	IF
	// NX5001_2
		DiagsRetain.DG_NX5001_2_tGeneral_bActiveDiagnostics OR
		DiagsRetain.DG_NX5001_2_tGeneral_bBusCommunicationError OR
		DiagsRetain.DG_NX5001_2_tGeneral_bConfigMismatch OR
		DiagsRetain.DG_NX5001_2_tGeneral_bFatalError OR
		DiagsRetain.DG_NX5001_2_tGeneral_bNX5001NoCfg OR
		DiagsRetain.DG_NX5001_2_tGeneral_bOTDSwitchError OR
		DiagsRetain.DG_NX5001_2_tGeneral_bPbusCommFail OR
		DiagsRetain.DG_NX5001_2_tGeneral_bSlaveNotConfigured OR
		DiagsRetain.DG_NX5001_2_tGeneral_bSlaveNotPresent OR
		DiagsRetain.DG_NX5001_2_tGeneral_bSlaveWithDiagnostic OR
		DiagsRetain.DG_NX5001_2_tGeneral_bStsEnableInterface OR
	//	DiagsRetain.DG_NX5001_2_tGeneral_bStsMstRedundEnable OR   Demanda 17571
		DiagsRetain.DG_NX5001_2_tGeneral_bWatchdogError THEN
   	 	bDiag_Error_NX5001_2:= TRUE;
	ELSE
		bDiag_Error_NX5001_2:= FALSE;	
	END_IF
	
	IF
	// NX5001_3
		DiagsRetain.DG_NX5001_3_tGeneral_bActiveDiagnostics OR
		DiagsRetain.DG_NX5001_3_tGeneral_bBusCommunicationError OR
		DiagsRetain.DG_NX5001_3_tGeneral_bConfigMismatch OR
		DiagsRetain.DG_NX5001_3_tGeneral_bFatalError OR
		DiagsRetain.DG_NX5001_3_tGeneral_bNX5001NoCfg OR
		DiagsRetain.DG_NX5001_3_tGeneral_bOTDSwitchError OR
		DiagsRetain.DG_NX5001_3_tGeneral_bPbusCommFail OR
		DiagsRetain.DG_NX5001_3_tGeneral_bSlaveNotConfigured OR
		DiagsRetain.DG_NX5001_3_tGeneral_bSlaveNotPresent OR
		DiagsRetain.DG_NX5001_3_tGeneral_bSlaveWithDiagnostic OR
		DiagsRetain.DG_NX5001_3_tGeneral_bStsEnableInterface OR
	//	DiagsRetain.DG_NX5001_3_tGeneral_bStsMstRedundEnable OR   Demanda 17571
		DiagsRetain.DG_NX5001_3_tGeneral_bWatchdogError THEN
  	 	bDiag_Error_NX5001_3:= TRUE;
	ELSE
		bDiag_Error_NX5001_3:= FALSE;	
	END_IF
	
	IF
	// NX5000_1	
		DiagsRetain.DG_NX5000_1_tGeneral_bActiveDiagnostics OR
		DiagsRetain.DG_NX5000_1_tGeneral_bBusCommunicationError OR
		DiagsRetain.DG_NX5000_1_tGeneral_bConfigMismatch OR
		DiagsRetain.DG_NX5000_1_tGeneral_bFatalError OR
		DiagsRetain.DG_NX5000_1_tGeneral_bOTDSwitchError OR
		DiagsRetain.DG_NX5000_1_tGeneral_bWatchdogError OR
		DiagsRetain.DG_NX5000_1_tNX5000_bNX5000NoCfg OR
		DiagsRetain.DG_NX5000_1_tNX5000_bStsEthLink THEN
    	bDiag_Error_NX5000_1:= TRUE;
	ELSE
		bDiag_Error_NX5000_1:= FALSE;	
	END_IF
	
	IF
	// NX5000_2	
		DiagsRetain.DG_NX5000_2_tGeneral_bActiveDiagnostics OR
		DiagsRetain.DG_NX5000_2_tGeneral_bBusCommunicationError OR
		DiagsRetain.DG_NX5000_2_tGeneral_bConfigMismatch OR
		DiagsRetain.DG_NX5000_2_tGeneral_bFatalError OR
		DiagsRetain.DG_NX5000_2_tGeneral_bOTDSwitchError OR
		DiagsRetain.DG_NX5000_2_tGeneral_bWatchdogError OR
		DiagsRetain.DG_NX5000_2_tNX5000_bNX5000NoCfg OR
		DiagsRetain.DG_NX5000_2_tNX5000_bStsEthLink THEN
    	bDiag_Error_NX5000_2:= TRUE;
	ELSE
		bDiag_Error_NX5000_2:= FALSE;	
	END_IF
	
	IF
	// NX5000_3	
		DiagsRetain.DG_NX5000_3_tGeneral_bActiveDiagnostics OR
		DiagsRetain.DG_NX5000_3_tGeneral_bBusCommunicationError OR
		DiagsRetain.DG_NX5000_3_tGeneral_bConfigMismatch OR
		DiagsRetain.DG_NX5000_3_tGeneral_bFatalError OR
		DiagsRetain.DG_NX5000_3_tGeneral_bOTDSwitchError OR
		DiagsRetain.DG_NX5000_3_tGeneral_bWatchdogError OR
		DiagsRetain.DG_NX5000_3_tNX5000_bNX5000NoCfg OR
		DiagsRetain.DG_NX5000_3_tNX5000_bStsEthLink THEN
    	bDiag_Error_NX5000_3:= TRUE;
	ELSE
		bDiag_Error_NX5000_3:= FALSE;	
	END_IF
	
	IF
	// DiagsRetain.DG_MODBUS_Master_1
		DiagsRetain.DG_MODBUS_Master_1_tDiag_bConfigFailure OR
		DiagsRetain.DG_MODBUS_Master_1_tDiag_bModuleFailure OR
		DiagsRetain.DG_MODBUS_Master_1_tDiag_bRXFailure OR
		DiagsRetain.DG_MODBUS_Master_1_tDiag_bTXFailure THEN
   	 	bDiag_Error_MODBUS_Master_1:= TRUE;
	ELSE
		bDiag_Error_MODBUS_Master_1:= FALSE;	
	END_IF
	
	IF
	// MODBUS_Slave_1	
		DiagsRetain.DG_MODBUS_Slave_1_tDiag_bConfigFailure OR
		DiagsRetain.DG_MODBUS_Slave_1_tDiag_bModuleFailure OR
		DiagsRetain.DG_MODBUS_Slave_1_tDiag_bRXFailure OR
		DiagsRetain.DG_MODBUS_Slave_1_tDiag_bTXFailure THEN
   		bDiag_Error_MODBUS_Slave_1:= TRUE;
	ELSE
		bDiag_Error_MODBUS_Slave_1:= FALSE;	
	END_IF
	
	IF
	// MODBUS_Client_2
		DiagsRetain.DG_MODBUS_Client_2_tDiag_bConfigFailure OR
//		DiagsRetain.DG_MODBUS_Client_2_tDiag_bModuleFailure OR 	// Demanda 13816
		DiagsRetain.DG_MODBUS_Client_2_tDiag_bRXFailure OR
		DiagsRetain.DG_MODBUS_Client_2_tDiag_bTXFailure THEN
    	bDiag_Error_MODBUS_Client_2:= TRUE;
	ELSE
		bDiag_Error_MODBUS_Client_2:= FALSE;	
	END_IF
	
	IF
	// MODBUS_Server_2
		DiagsRetain.DG_MODBUS_Server_2_tDiag_bConfigFailure OR
		DiagsRetain.DG_MODBUS_Server_2_tDiag_bModuleFailure OR
		DiagsRetain.DG_MODBUS_Server_2_tDiag_bRXFailure OR
		DiagsRetain.DG_MODBUS_Server_2_tDiag_bTXFailure THEN
    	bDiag_Error_MODBUS_Server_2:= TRUE;
	ELSE
		bDiag_Error_MODBUS_Server_2:= FALSE;	
	END_IF
	
	IF
	// MODBUS_Client_3
		DiagsRetain.DG_MODBUS_Client_3_tDiag_bConfigFailure OR
		DiagsRetain.DG_MODBUS_Client_3_tDiag_bModuleFailure OR
		DiagsRetain.DG_MODBUS_Client_3_tDiag_bRXFailure OR
		DiagsRetain.DG_MODBUS_Client_3_tDiag_bTXFailure THEN
    	bDiag_Error_MODBUS_Client_3:= TRUE;
	ELSE
		bDiag_Error_MODBUS_Client_3:= FALSE;	
	END_IF
	
	IF
	// MODBUS_Server_3
		DiagsRetain.DG_MODBUS_Server_3_tDiag_bConfigFailure OR
//		DiagsRetain.DG_MODBUS_Server_3_tDiag_bModuleFailure OR  	// Demanda 13816
		DiagsRetain.DG_MODBUS_Server_3_tDiag_bRXFailure OR
		DiagsRetain.DG_MODBUS_Server_3_tDiag_bTXFailure THEN
    	bDiag_Error_MODBUS_Server_3:= TRUE;
	ELSE
		bDiag_Error_MODBUS_Server_3:= FALSE;	
	END_IF
	
	IF
	// MODBUS_Client_4
		DiagsRetain.DG_MODBUS_Client_4_tDiag_bConfigFailure OR
		DiagsRetain.DG_MODBUS_Client_4_tDiag_bModuleFailure OR
		DiagsRetain.DG_MODBUS_Client_4_tDiag_bRXFailure OR
		DiagsRetain.DG_MODBUS_Client_4_tDiag_bTXFailure THEN
    	bDiag_Error_MODBUS_Client_4:= TRUE;
	ELSE
		bDiag_Error_MODBUS_Client_4:= FALSE;	
	END_IF
	
	IF
	// MODBUS_Server_4	
		DiagsRetain.DG_MODBUS_Server_4_tDiag_bConfigFailure OR
//		DiagsRetain.DG_MODBUS_Server_4_tDiag_bModuleFailure OR  	// Demanda 13816
		DiagsRetain.DG_MODBUS_Server_4_tDiag_bRXFailure OR
		DiagsRetain.DG_MODBUS_Server_4_tDiag_bTXFailure THEN
    	bDiag_Error_MODBUS_Server_4:= TRUE;
	ELSE
		bDiag_Error_MODBUS_Server_4:= FALSE;	
	END_IF
	

	IF		
		//PO1000
		DiagsRetain.DG_REM05_PO1000_bHardwareFailure OR
		DiagsRetain.DG_REM05_PO1000_bPowerSupplyFail THEN
	   	bDiag_Error_PO1000_REM05:= TRUE;
	ELSE
		bDiag_Error_PO1000_REM05:= FALSE;	
	END_IF
	
	IF		
		//PO2020
		DiagsRetain.DG_REM05_PO2020_bHardwareFailure OR
		DiagsRetain.DG_REM05_PO2020_bPowerSupplyFail THEN
		bDiag_Error_PO2020_REM05:= TRUE;
	ELSE
		bDiag_Error_PO2020_REM05:= FALSE;	
	END_IF

	IF		
		//PO9100	
		DiagsRetain.DG_REM05_PO9100_bReserved00 THEN
		bDiag_Error_PO9100_REM05:= TRUE;
	ELSE
		bDiag_Error_PO9100_REM05:= FALSE;	
	END_IF	
	
	IF		
	//PO1212
	DiagsRetain.DG_REM10_PO1212_bFuseOpen OR
	DiagsRetain.DG_REM10_PO1212_bHardwareFailure OR
	DiagsRetain.DG_REM10_PO1212_bNoParametrizedModule OR
	DiagsRetain.DG_REM10_PO1212_bOverTemp OR
	DiagsRetain.DG_REM10_PO1212_aCh0_bOpenSensor OR
	DiagsRetain.DG_REM10_PO1212_aCh0_bOverRange OR
	DiagsRetain.DG_REM10_PO1212_aCh0_bSensorShortCircuit OR
	DiagsRetain.DG_REM10_PO1212_aCh0_bWrongParameters OR
	DiagsRetain.DG_REM10_PO1212_aCh1_bOpenSensor OR
	DiagsRetain.DG_REM10_PO1212_aCh1_bOverRange OR
	DiagsRetain.DG_REM10_PO1212_aCh1_bSensorShortCircuit OR
	DiagsRetain.DG_REM10_PO1212_aCh1_bWrongParameters OR
	DiagsRetain.DG_REM10_PO1212_aCh2_bOpenSensor OR
	DiagsRetain.DG_REM10_PO1212_aCh2_bOverRange OR
	DiagsRetain.DG_REM10_PO1212_aCh2_bSensorShortCircuit OR
	DiagsRetain.DG_REM10_PO1212_aCh2_bWrongParameters OR
	DiagsRetain.DG_REM10_PO1212_aCh3_bOpenSensor OR
	DiagsRetain.DG_REM10_PO1212_aCh3_bOverRange OR
	DiagsRetain.DG_REM10_PO1212_aCh3_bSensorShortCircuit OR
	DiagsRetain.DG_REM10_PO1212_aCh3_bWrongParameters OR
	DiagsRetain.DG_REM10_PO1212_aCh4_bOpenSensor OR
	DiagsRetain.DG_REM10_PO1212_aCh4_bOverRange OR
	DiagsRetain.DG_REM10_PO1212_aCh4_bSensorShortCircuit OR
	DiagsRetain.DG_REM10_PO1212_aCh4_bWrongParameters OR
	DiagsRetain.DG_REM10_PO1212_aCh5_bOpenSensor OR
	DiagsRetain.DG_REM10_PO1212_aCh5_bOverRange OR
	DiagsRetain.DG_REM10_PO1212_aCh5_bSensorShortCircuit OR
	DiagsRetain.DG_REM10_PO1212_aCh5_bWrongParameters OR
	DiagsRetain.DG_REM10_PO1212_aCh6_bOpenSensor OR
	DiagsRetain.DG_REM10_PO1212_aCh6_bOverRange OR
	DiagsRetain.DG_REM10_PO1212_aCh6_bSensorShortCircuit OR
	DiagsRetain.DG_REM10_PO1212_aCh6_bWrongParameters OR
	DiagsRetain.DG_REM10_PO1212_aCh7_bOpenSensor OR
	DiagsRetain.DG_REM10_PO1212_aCh7_bOverRange OR
	DiagsRetain.DG_REM10_PO1212_aCh7_bSensorShortCircuit OR
	DiagsRetain.DG_REM10_PO1212_aCh7_bWrongParameters THEN
		bDiag_Error_PO1212_REM10:= TRUE;
	ELSE
		bDiag_Error_PO1212_REM10:= FALSE;	
	END_IF		
	
	IF		
	//PO2132
	DiagsRetain.DG_REM10_PO2132_bNoParametrizedModule OR
	DiagsRetain.DG_REM10_PO2132_bPowerSupplyFail OR
	DiagsRetain.DG_REM10_PO2132_aCh0_bOpenSensor OR
	DiagsRetain.DG_REM10_PO2132_aCh0_bWrongParameters OR
	DiagsRetain.DG_REM10_PO2132_aCh1_bOpenSensor OR
	DiagsRetain.DG_REM10_PO2132_aCh1_bWrongParameters OR
	DiagsRetain.DG_REM10_PO2132_aCh2_bOpenSensor OR
	DiagsRetain.DG_REM10_PO2132_aCh2_bWrongParameters OR
	DiagsRetain.DG_REM10_PO2132_aCh3_bOpenSensor OR
	DiagsRetain.DG_REM10_PO2132_aCh3_bWrongParameters THEN
		bDiag_Error_PO2132_REM10:= TRUE;
	ELSE
		bDiag_Error_PO2132_REM10:= FALSE;	
	END_IF		
	
	IF		
	//PO9100
	DiagsRetain.DG_REM10_PO9100_bReserved00 THEN
			bDiag_Error_PO9100_REM10:= TRUE;
	ELSE
		bDiag_Error_PO9100_REM10:= FALSE;	
	END_IF	
	
	IF		
	//PO1000
	DiagsRetain.DG_REM04_PO1000_bHardwareFailure OR
	DiagsRetain.DG_REM04_PO1000_bPowerSupplyFail THEN
		bDiag_Error_PO1000_REM04:= TRUE;
	ELSE
		bDiag_Error_PO1000_REM04:= FALSE;	
	END_IF	

	
	IF 
		bDiag_Error_NX3030 OR
		bDiag_Error_NX4010 OR
		bDiag_Error_NX5001_1 OR
		bDiag_Error_NX5001_2 OR
		bDiag_Error_NX5001_3 OR
		bDiag_Error_NX5000_1 OR
		bDiag_Error_NX5000_2 OR
		bDiag_Error_NX5000_3 OR
		bDiag_Error_MODBUS_Master_1 OR
		bDiag_Error_MODBUS_Slave_1 OR
		bDiag_Error_MODBUS_Client_2 OR
		bDiag_Error_MODBUS_Server_2 OR
		bDiag_Error_MODBUS_Client_3 OR
		bDiag_Error_MODBUS_Server_3 OR
		bDiag_Error_MODBUS_Client_4 OR
		bDiag_Error_MODBUS_Server_4 OR	
		bDiag_Error_PO1000_REM05 OR
		bDiag_Error_PO2020_REM05 OR
		bDiag_Error_PO9100_REM05 OR
		bDiag_Error_PO1212_REM10 OR
		bDiag_Error_PO2132_REM10 OR
		bDiag_Error_PO9100_REM10 OR
		bDiag_Error_PO1000_REM04 THEN
		PersistentVars.bActiveDiagPlcB:= TRUE;
	ELSE
		PersistentVars.bActiveDiagPlcB:= FALSE;
	END_IF
END_IF	

// Limpa diagnóstico com um comando de CleanTest
IF SymbolicsNonRedundant.bEnableCleanStats_CheckDiagsRetain THEN
	SymbolicsNonRedundant.bEnableCleanStats_CheckDiagsRetain:= FALSE;
	PersistentVars.bActiveDiagPlcB:= FALSE;
	PersistentVars.bActiveDiagPlcA:= FALSE;
	/// Depuração 1
	auiDebugRedDataSync[0]:= auiDebugRedForceSync[0]:= 0;
	auiDebugRedDataSync[1]:= auiDebugRedForceSync[1]:= 0;
	auiDebugRedDataSync[2]:= auiDebugRedForceSync[2]:= 0;
	auiDebugRedDataSync[3]:= auiDebugRedForceSync[3]:= 0;
	auiDebugRedDataSync[4]:= auiDebugRedForceSync[4]:= 0;
	auiDebugRedDataSync[5]:= auiDebugRedForceSync[5]:= 0;
	auiDebugRedDataSync[6]:= auiDebugRedForceSync[6]:= 0;
END_IF

/// Depuração 2
IF NOT DG_NX4010.tRedundancy.RedDgnLoc.sGeneral_Diag.bRedDataSync THEN
	CASE fbRedundancyManagement.m_fbDiagnosticsLocal.eRedState OF
		REDUNDANCY_STATE.NOT_CONFIGURED:	auiDebugRedDataSync[0]:= MIN(auiDebugRedDataSync[0] + 1, 65000);
		REDUNDANCY_STATE.INIT:				auiDebugRedDataSync[1]:= MIN(auiDebugRedDataSync[1] + 1, 65000);
		REDUNDANCY_STATE.STARTING:			auiDebugRedDataSync[2]:= MIN(auiDebugRedDataSync[2] + 1, 65000);
		REDUNDANCY_STATE.STANDBY:			auiDebugRedDataSync[3]:= MIN(auiDebugRedDataSync[3] + 1, 65000);
		REDUNDANCY_STATE.ACTIVE:			auiDebugRedDataSync[4]:= MIN(auiDebugRedDataSync[4] + 1, 65000);
		REDUNDANCY_STATE.INACTIVE:			auiDebugRedDataSync[5]:= MIN(auiDebugRedDataSync[5] + 1, 65000);
	ELSE
		auiDebugRedDataSync[6]:= MIN(auiDebugRedDataSync[6] + 1, 65000);
	END_CASE
END_IF

/// Depuração 3
IF NOT DG_NX4010.tRedundancy.RedDgnLoc.sGeneral_Diag.bRedForceSync THEN
	CASE fbRedundancyManagement.m_fbDiagnosticsLocal.eRedState OF
		REDUNDANCY_STATE.NOT_CONFIGURED:	auiDebugRedForceSync[0]:= MIN(auiDebugRedForceSync[0] + 1, 65000);
		REDUNDANCY_STATE.INIT:				auiDebugRedForceSync[1]:= MIN(auiDebugRedForceSync[1] + 1, 65000);
		REDUNDANCY_STATE.STARTING:			auiDebugRedForceSync[2]:= MIN(auiDebugRedForceSync[2] + 1, 65000);
		REDUNDANCY_STATE.STANDBY:			auiDebugRedForceSync[3]:= MIN(auiDebugRedForceSync[3] + 1, 65000);
		REDUNDANCY_STATE.ACTIVE:			auiDebugRedForceSync[4]:= MIN(auiDebugRedForceSync[4] + 1, 65000);
		REDUNDANCY_STATE.INACTIVE:			auiDebugRedForceSync[5]:= MIN(auiDebugRedForceSync[5] + 1, 65000);
	ELSE
		auiDebugRedForceSync[6]:= MIN(auiDebugRedForceSync[6] + 1, 65000);
	END_CASE
END_IF

// Registra o tempo do sistema
SysTimeGetUs(uliPouEndTime);
// Calcula duração mínima/máxima desta POU
MinMaxTimes.uliPouMinTime_CheckDiags:= MIN(MinMaxTimes.uliPouMinTime_CheckDiags, uliPouEndTime - uliPouIniTime);
MinMaxTimes.uliPouMaxTime_CheckDiags:= MAX(MinMaxTimes.uliPouMaxTime_CheckDiags, uliPouEndTime - uliPouIniTime);

END_PROGRAM

// Device/Application/UserPOUs/Non-Redundant/DaylightSavingTime
PROGRAM DaylightSavingTime
VAR
	xDateAndTime:	EXTENDED_DATE_AND_TIME;
	byDayOfWeek:	BYTE;
	xTimeZoneRd:	TIMEZONESETTINGS;
	xTimeZoneWr:	TIMEZONESETTINGS;
	// Array de referência para cada ano:
	// 14 indica que o terceiro domingo do mês de fevereiro NÃO coincide com o carnaval
	// 21 indica que o terceiro domingo do mês de fevereiro coincide com o carnaval
	aby3rd4thDay:	ARRAY[2017..2027] OF BYTE:= [14,14,14,14,14,14,21,14,14,21,14];
	// Contador de escritas do timezone em função do início/fim do horário de verão
	// (configurar o parâmetro "HX3040 > Synchronism > Time Zone" para o valor -3:00) 
	// (se iniciar a aplicação no horário de verão, o contador vai para 1 na partida) 
	udiTZWriteCnt:	UDINT;
	uliPouIniTime:	ULINT;
	uliPouEndTime:	ULINT;
END_VAR

// Rotina que detecta se é horário de verão, ajustando o timezone da UCP se necessário.

// Registra o tempo do sistema
SysTimeGetUs(uliPouIniTime);

// Leitura da data e hora atual, com sucesso...
IF NextoStandard.GetDateAndTime(xDateAndTime) = 0 THEN
	
	// Leitura do dia da semana
	byDayOfWeek:= NextoStandard.GetDayOfWeek();
	
	// Segundo o decreto presidencial 6.558 de 08/09/2008, o horário de verão inicia
	// no terceiro domingo do mês de outubro e termina no terceiro domingo do mês de
	// fevereiro (ou quarto, se o terceiro coincidir com a semana do carnaval)
	IF 	(xDateAndTime.byMonth = 10 AND (xDateAndTime.byDayOfMonth >= 14 + byDayOfWeek)) OR
		(xDateAndTime.byMonth = 11) OR
		(xDateAndTime.byMonth = 12) OR
		(xDateAndTime.byMonth = 1) OR
		(xDateAndTime.byMonth = 2 AND (xDateAndTime.byDayOfMonth < aby3rd4thDay[xDateAndTime.wYear] + byDayOfWeek)) THEN
			// Indica que é horário de verão
			NonRedData.bDaylightSavingTime:= TRUE;
	ELSE
			// Indica que NÃO é horário de verão
			NonRedData.bDaylightSavingTime:= FALSE;
	END_IF
	
	// Leitura do timezone, com sucesso...
	IF NextoStandard.GetTimeZone(xTimeZoneRd) = 0 THEN
		// Se horário de verão, timezone deve ser -2:00, caso contrário deve ser -3:00
		// Dispara um comando de escrita do timezone se encontrar alguma divergência
		IF 	(NonRedData.bDaylightSavingTime = TRUE AND (xTimeZoneRd.iHour <> -2 OR xTimeZoneRd.iMinutes <> 0)) OR
			(NonRedData.bDaylightSavingTime = FALSE AND (xTimeZoneRd.iHour <> -3 OR xTimeZoneRd.iMinutes <> 0)) THEN
				// Ajusta timezone para horário de verão ou horário normal
				IF NonRedData.bDaylightSavingTime = TRUE THEN
					xTimeZoneWr.iHour:= -2;
					xTimeZoneWr.iMinutes:= 0;
				ELSE
					xTimeZoneWr.iHour:= -3;
					xTimeZoneWr.iMinutes:= 0;
				END_IF
				// Chama função de escrita do timezone
				NextoStandard.SetTimeZone(xTimeZoneWr);
				// Incrementa o contador de escritas do timezone
				udiTZWriteCnt:= udiTZWriteCnt + 1;
		END_IF
	END_IF

END_IF

// Registra o tempo do sistema
SysTimeGetUs(uliPouEndTime);
// Calcula duração mínima/máxima desta POU
MinMaxTimes.uliPouMinTime_DaylightSavingTime:= MIN(MinMaxTimes.uliPouMinTime_DaylightSavingTime, uliPouEndTime - uliPouIniTime);
MinMaxTimes.uliPouMaxTime_DaylightSavingTime:= MAX(MinMaxTimes.uliPouMaxTime_DaylightSavingTime, uliPouEndTime - uliPouIniTime);

END_PROGRAM

// Device/Application/UserPOUs/Non-Redundant/CheckSpecialVarsRed
PROGRAM CheckSpecialVarsRed
VAR
	bPulse_100ms:		BOOL;
	bPulse_500ms:		BOOL;
	bPulse_1s:			BOOL;
	bPulse_2s:			BOOL;
	bPulse_5s:			BOOL;
	bPulse_10s:			BOOL;
	bPulse_30s:			BOOL;
	bPulse_60s:			BOOL;
	bPulse_Scan:		BOOL;
	
	di100msTimer:		DINT;
	di500msTimer:		DINT;
	di1sTimer:			DINT;
	di2sTimer:			DINT;
	di5sTimer:			DINT;
	di10sTimer:			DINT;
	di30sTimer:			DINT;
	di60sTimer:			DINT;
	
	bPulse100msFail:	BOOL;
	bPulse500msFail:	BOOL;
	bPulse1sFail:		BOOL;
	bPulse2sFail:		BOOL;
	bPulse5sFail:		BOOL;
	bPulse10sFail:		BOOL;
	bPulse30sFail:		BOOL;
	bPulse60sFail:		BOOL;
	bPulseScanFail:		BOOL;
	
	diMainTaskIntervalGapMs:	DINT:= ProjectConstants.iMainTaskInterval * 3 / 2;
	
	uliPouMemTime: 				ULINT;
	
END_VAR

// 
// POU para consistência das variáveis especiais redundantes.
// Esta POU deve ser chamada pela POU CheckSpecialVariables.
// 

// Detecta quando a tarefa cíclica deixou de ser chamada por um ciclo
// (com 10% de folga devido ao jitter negativo da tarefa)
// (também converte de milisegundos para microsegundos)
IF CheckSpecialVariables.uliPouIniTime > uliPouMemTime + DINT_TO_ULINT(ProjectConstants.iMainTaskInterval * 1900) THEN
	// Quando isso acontece, algumas variáveis de temporização e controle precisam ser ajustadas
	di100msTimer:= UDINT_TO_DINT(SpecialVariablesRedundantPrg.udiMicroAcc MOD 50000) / 1000;
	di500msTimer:= UDINT_TO_DINT(SpecialVariablesRedundantPrg.udiMicroAcc MOD 250000) / 1000;
	di1sTimer:= UDINT_TO_DINT(SpecialVariablesRedundantPrg.udiMicroAcc MOD 500000) / 1000;
	di2sTimer:= UDINT_TO_DINT(SpecialVariablesRedundantPrg.udiMicroAcc MOD 1000000) / 1000;
	di5sTimer:= UDINT_TO_DINT(SpecialVariablesRedundantPrg.udiMicroAcc MOD 2500000) / 1000;
	di10sTimer:= UDINT_TO_DINT(SpecialVariablesRedundantPrg.udiMicroAcc MOD 5000000) / 1000;
	di30sTimer:= UDINT_TO_DINT(SpecialVariablesRedundantPrg.udiMicroAcc MOD 15000000) / 1000;
	di60sTimer:= UDINT_TO_DINT(SpecialVariablesRedundantPrg.udiMicroAcc MOD 30000000) / 1000;
	bPulse_100ms:= Special_Variables_Redundant.Pulse_100ms_Redundant;
	bPulse_500ms:= Special_Variables_Redundant.Pulse_500ms_Redundant;
	bPulse_1s:= Special_Variables_Redundant.Pulse_1s_Redundant;
	bPulse_2s:= Special_Variables_Redundant.Pulse_2s_Redundant;
	bPulse_5s:= Special_Variables_Redundant.Pulse_5s_Redundant;
	bPulse_10s:= Special_Variables_Redundant.Pulse_10s_Redundant;
	bPulse_30s:= Special_Variables_Redundant.Pulse_30s_Redundant;
	bPulse_60s:= Special_Variables_Redundant.Pulse_60s_Redundant;
	bPulse_Scan:= NOT Special_Variables_Redundant.Pulse_Scan_Redundant;
END_IF
// Memoriza o tempo de ciclo atual
uliPouMemTime:= CheckSpecialVariables.uliPouIniTime;

// Executa parte do mesmo código que a SpecialVariablesRedundantPrg(), porém com variáveis locais:

	// Update scan pulse
	bPulse_Scan:= NOT bPulse_Scan;
	
// Mede e consiste a duração dos pulsos: frequência e duty-cycle (50%)

// Consiste o pulso de 100ms se o intervalo da tarefa não exceder os 33%
IF 100 > 3 * ProjectConstants.iMainTaskInterval THEN
	// Se o sinal não mudou de estado...
	IF bPulse_100ms = Special_Variables_Redundant.Pulse_100ms_Redundant THEN
		// Atualiza temporizador do sinal
		di100msTimer:= di100msTimer + ProjectConstants.iMainTaskInterval;
		// Indica erro caso o sinal não tenha mudado de estado no dobro do tempo esperado
		IF di100msTimer > 100 THEN bPulse100msFail:= TRUE; END_IF
	// Se o sinal mudou de estado...
	ELSE
		// Indica erro caso o sinal tenha mudado de estado antes ou depois do tempo esperado
		IF	di100msTimer < (100 / 2 - diMainTaskIntervalGapMs) OR
			di100msTimer > (100 / 2 + diMainTaskIntervalGapMs) THEN
				bPulse100msFail:= TRUE;
		END_IF
		// Inicializa o temporizador do sinal
		di100msTimer:= ProjectConstants.iMainTaskInterval;
		// Memoriza o estado atual do sinal
		bPulse_100ms:= Special_Variables_Redundant.Pulse_100ms_Redundant;
	END_IF
END_IF

// Consiste o pulso de 500ms se o intervalo da tarefa não exceder os 33%
IF 500 > 3 * ProjectConstants.iMainTaskInterval THEN
	// Se o sinal não mudou de estado...
	IF bPulse_500ms = Special_Variables_Redundant.Pulse_500ms_Redundant THEN
		// Atualiza temporizador do sinal
		di500msTimer:= di500msTimer + ProjectConstants.iMainTaskInterval;
		// Indica erro caso o sinal não tenha mudado de estado no dobro do tempo esperado
		IF di500msTimer > 500 THEN bPulse500msFail:= TRUE; END_IF
	// Se o sinal mudou de estado...
	ELSE
		// Indica erro caso o sinal tenha mudado de estado antes ou depois do tempo esperado
		IF	di500msTimer < (500 / 2 - diMainTaskIntervalGapMs) OR
			di500msTimer > (500 / 2 + diMainTaskIntervalGapMs) THEN
				bPulse500msFail:= TRUE;
		END_IF
		// Inicializa o temporizador do sinal
		di500msTimer:= ProjectConstants.iMainTaskInterval;
		// Memoriza o estado atual do sinal
		bPulse_500ms:= Special_Variables_Redundant.Pulse_500ms_Redundant;
	END_IF
END_IF

// Se o sinal não mudou de estado...
IF bPulse_1s = Special_Variables_Redundant.Pulse_1s_Redundant THEN
	// Atualiza temporizador do sinal
	di1sTimer:= di1sTimer + ProjectConstants.iMainTaskInterval;
	// Indica erro caso o sinal não tenha mudado de estado no dobro do tempo esperado
	IF di1sTimer > 1000 THEN bPulse1sFail:= TRUE; END_IF
// Se o sinal mudou de estado...
ELSE
	// Indica erro caso o sinal tenha mudado de estado antes ou depois do tempo esperado
	IF	di1sTimer < (1000 / 2 - diMainTaskIntervalGapMs) OR
		di1sTimer > (1000 / 2 + diMainTaskIntervalGapMs) THEN
			bPulse1sFail:= TRUE;
	END_IF
	// Inicializa o temporizador do sinal
	di1sTimer:= ProjectConstants.iMainTaskInterval;
	// Memoriza o estado atual do sinal
	bPulse_1s:= Special_Variables_Redundant.Pulse_1s_Redundant;
END_IF

// Se o sinal não mudou de estado...
IF bPulse_2s = Special_Variables_Redundant.Pulse_2s_Redundant THEN
	// Atualiza temporizador do sinal
	di2sTimer:= di2sTimer + ProjectConstants.iMainTaskInterval;
	// Indica erro caso o sinal não tenha mudado de estado no dobro do tempo esperado
	IF di2sTimer > 2000 THEN bPulse2sFail:= TRUE; END_IF
// Se o sinal mudou de estado...
ELSE
	// Indica erro caso o sinal tenha mudado de estado antes ou depois do tempo esperado
	IF	di2sTimer < (2000 / 2 - diMainTaskIntervalGapMs) OR
		di2sTimer > (2000 / 2 + diMainTaskIntervalGapMs) THEN
			bPulse2sFail:= TRUE;
	END_IF
	// Inicializa o temporizador do sinal
	di2sTimer:= ProjectConstants.iMainTaskInterval;
	// Memoriza o estado atual do sinal
	bPulse_2s:= Special_Variables_Redundant.Pulse_2s_Redundant;
END_IF

// Se o sinal não mudou de estado...
IF bPulse_5s = Special_Variables_Redundant.Pulse_5s_Redundant THEN
	// Atualiza temporizador do sinal
	di5sTimer:= di5sTimer + ProjectConstants.iMainTaskInterval;
	// Indica erro caso o sinal não tenha mudado de estado no dobro do tempo esperado
	IF di5sTimer > 5000 THEN bPulse5sFail:= TRUE; END_IF
// Se o sinal mudou de estado...
ELSE
	// Indica erro caso o sinal tenha mudado de estado antes ou depois do tempo esperado
	IF	di5sTimer < (5000 / 2 - diMainTaskIntervalGapMs) OR
		di5sTimer > (5000 / 2 + diMainTaskIntervalGapMs) THEN
			bPulse5sFail:= TRUE;
	END_IF
	// Inicializa o temporizador do sinal
	di5sTimer:= ProjectConstants.iMainTaskInterval;
	// Memoriza o estado atual do sinal
	bPulse_5s:= Special_Variables_Redundant.Pulse_5s_Redundant;
END_IF

// Se o sinal não mudou de estado...
IF bPulse_10s = Special_Variables_Redundant.Pulse_10s_Redundant THEN
	// Atualiza temporizador do sinal
	di10sTimer:= di10sTimer + ProjectConstants.iMainTaskInterval;
	// Indica erro caso o sinal não tenha mudado de estado no dobro do tempo esperado
	IF di10sTimer > 10000 THEN bPulse10sFail:= TRUE; END_IF
// Se o sinal mudou de estado...
ELSE
	// Indica erro caso o sinal tenha mudado de estado antes ou depois do tempo esperado
	IF	di10sTimer < (10000 / 2 - diMainTaskIntervalGapMs) OR
		di10sTimer > (10000 / 2 + diMainTaskIntervalGapMs) THEN
			bPulse10sFail:= TRUE;
	END_IF
	// Inicializa o temporizador do sinal
	di10sTimer:= ProjectConstants.iMainTaskInterval;
	// Memoriza o estado atual do sinal
	bPulse_10s:= Special_Variables_Redundant.Pulse_10s_Redundant;
END_IF

// Se o sinal não mudou de estado...
IF bPulse_30s = Special_Variables_Redundant.Pulse_30s_Redundant THEN
	// Atualiza temporizador do sinal
	di30sTimer:= di30sTimer + ProjectConstants.iMainTaskInterval;
	// Indica erro caso o sinal não tenha mudado de estado no dobro do tempo esperado
	IF di30sTimer > 30000 THEN bPulse30sFail:= TRUE; END_IF
// Se o sinal mudou de estado...
ELSE
	// Indica erro caso o sinal tenha mudado de estado antes ou depois do tempo esperado
	IF	di30sTimer < (30000 / 2 - diMainTaskIntervalGapMs) OR
		di30sTimer > (30000 / 2 + diMainTaskIntervalGapMs) THEN
			bPulse30sFail:= TRUE;
	END_IF
	// Inicializa o temporizador do sinal
	di30sTimer:= ProjectConstants.iMainTaskInterval;
	// Memoriza o estado atual do sinal
	bPulse_30s:= Special_Variables_Redundant.Pulse_30s_Redundant;
END_IF

// Se o sinal não mudou de estado...
IF bPulse_60s = Special_Variables_Redundant.Pulse_60s_Redundant THEN
	// Atualiza temporizador do sinal
	di60sTimer:= di60sTimer + ProjectConstants.iMainTaskInterval;
	// Indica erro caso o sinal não tenha mudado de estado no dobro do tempo esperado
	IF di60sTimer > 60000 THEN bPulse60sFail:= TRUE; END_IF
// Se o sinal mudou de estado...
ELSE
	// Indica erro caso o sinal tenha mudado de estado antes ou depois do tempo esperado
	IF	di60sTimer < (60000 / 2 - diMainTaskIntervalGapMs) OR
		di60sTimer > (60000 / 2 + diMainTaskIntervalGapMs) THEN
			bPulse60sFail:= TRUE;
	END_IF
	// Inicializa o temporizador do sinal
	di60sTimer:= ProjectConstants.iMainTaskInterval;
	// Memoriza o estado atual do sinal
	bPulse_60s:= Special_Variables_Redundant.Pulse_60s_Redundant;
END_IF

// Realiza as consistências para identificar falhas nos demais sinais da GVL Special_Variables
bPulseScanFail:= bPulseScanFail OR Special_Variables_Redundant.Pulse_Scan_Redundant <> bPulse_Scan;

END_PROGRAM

// Device/Application/SystemPOUs/SpecialVariablesRedundantPrg
(*This POU is blocked to edit.*)
{attribute 'hide'}
PROGRAM SpecialVariablesRedundantPrg
VAR
	udiMicroAcc:	UDINT;			// Microseconds accumulator
END_VAR

// Update pulse bits
IF SpecialVariablesPrg.uliLastSysTime > 0 THEN udiMicroAcc:= udiMicroAcc + ULINT_TO_UDINT(SpecialVariablesPrg.uliSystemTime - SpecialVariablesPrg.uliLastSysTime); END_IF
IF udiMicroAcc MOD 100000 >= 50000 THEN Pulse_100ms_Redundant:= TRUE; ELSE Pulse_100ms_Redundant:= FALSE; END_IF
IF udiMicroAcc MOD 500000 >= 250000 THEN Pulse_500ms_Redundant:= TRUE; ELSE Pulse_500ms_Redundant:= FALSE; END_IF
IF udiMicroAcc MOD 1000000 >= 500000 THEN Pulse_1s_Redundant:= TRUE; ELSE Pulse_1s_Redundant:= FALSE; END_IF
IF udiMicroAcc MOD 2000000 >= 1000000 THEN Pulse_2s_Redundant:= TRUE; ELSE Pulse_2s_Redundant:= FALSE; END_IF
IF udiMicroAcc MOD 5000000 >= 2500000 THEN Pulse_5s_Redundant:= TRUE; ELSE Pulse_5s_Redundant:= FALSE; END_IF
IF udiMicroAcc MOD 10000000 >= 5000000 THEN Pulse_10s_Redundant:= TRUE; ELSE Pulse_10s_Redundant:= FALSE; END_IF
IF udiMicroAcc MOD 30000000 >= 15000000 THEN Pulse_30s_Redundant:= TRUE; ELSE Pulse_30s_Redundant:= FALSE; END_IF
IF udiMicroAcc MOD 60000000 >= 30000000 THEN Pulse_60s_Redundant:= TRUE; ELSE Pulse_60s_Redundant:= FALSE; END_IF
udiMicroAcc:= udiMicroAcc MOD 120000000;

// Update scan pulse
Pulse_Scan_Redundant:= NOT Pulse_Scan_Redundant;

END_PROGRAM

// Device/Application/UserFunctions/CONCATENA_2WORD_TO_DWORD
FUNCTION CONCATENA_2WORD_TO_DWORD : DWORD
VAR_INPUT
	wWordHigh:	WORD;
	wWordLow:	WORD;
END_VAR
VAR
	dwWordHigh:		DWORD;
	dwNewHordHigh:	DWORD;
END_VAR

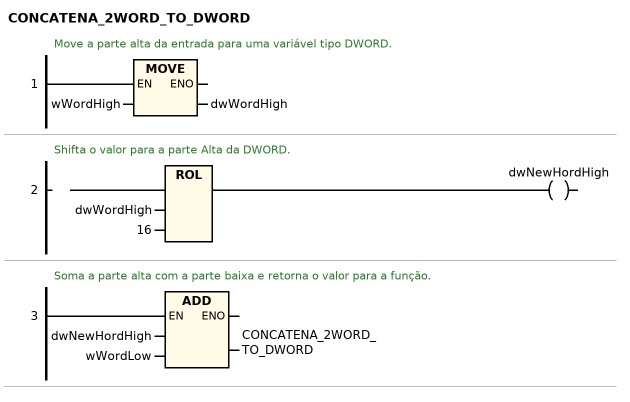
// NETWORK 1
// Move a parte alta da entrada para uma variável tipo DWORD.
dwWordHigh := wWordHigh;

// NETWORK 2
// Shifta o valor para a parte Alta da DWORD.
dwNewHordHigh := ROL(dwWordHigh, 16);

// NETWORK 3
// Soma a parte alta com a parte baixa e retorna o valor para a função.
CONCATENA_2WORD_TO_DWORD := dwNewHordHigh + wWordLow;

END_FUNCTION

// Device/Application/UserFunctions/iCounterIncFun
FUNCTION iCounterIncFun : INT
VAR_INPUT
	iCounter:	INT;
END_VAR
VAR
END_VAR

// Função para incrementar um contador até o valor limite codificado.
IF iCounter < ProjectConstants.iFailCounterLimit THEN
	iCounterIncFun:= iCounter + 1;
ELSE
	iCounterIncFun:= iCounter + 0;
END_IF

END_FUNCTION

// Library Information/GetLibVersion
// This function has been automatically generated from the project information.
FUNCTION GetLibVersion : VERSION
VAR_INPUT
	
END_VAR

GetLibVersion.uiMajor := 3;
GetLibVersion.uiMinor := 61;
GetLibVersion.uiServicePack := 0;
GetLibVersion.uiPatch := 0;

END_FUNCTION

// Library Information/GetLibVersionNumber
// This function has been automatically generated from the project information.
FUNCTION GetLibVersionNumber : DWORD
VAR_INPUT
	
END_VAR

GetLibVersionNumber := 54329344;

END_FUNCTION

// Library Information/IsLibReleased
// This function has been automatically generated from the project information.
FUNCTION IsLibReleased : BOOL
VAR_INPUT
	
END_VAR

IsLibReleased := FALSE;

END_FUNCTION

// Project Information/GetCompany
// This function has been automatically generated from the project information.
{attribute 'signature_flag' := '1073741824'}
{attribute 'register_in_runtime'}
FUNCTION GetCompany : WSTRING
VAR_INPUT
	
END_VAR

GetCompany := "Altus S.A.";

END_FUNCTION

// Project Information/GetTitle
// This function has been automatically generated from the project information.
{attribute 'signature_flag' := '1073741824'}
{attribute 'register_in_runtime'}
FUNCTION GetTitle : WSTRING
VAR_INPUT
	
END_VAR

GetTitle := "Super Teste NX3030";

END_FUNCTION

// Project Information/GetVersion
// This function has been automatically generated from the project information.
{attribute 'signature_flag' := '1073741824'}
{attribute 'register_in_runtime'}
FUNCTION GetVersion : VERSION
VAR_INPUT
	
END_VAR

GetVersion.uiMajor := 3;
GetVersion.uiMinor := 61;
GetVersion.uiServicePack := 0;
GetVersion.uiPatch := 0;

END_FUNCTION

// Project Information/GetTextProperty
// This function has been automatically generated from the project information.
{attribute 'signature_flag' := '1073741824'}
{attribute 'register_in_runtime'}
FUNCTION GetTextProperty : WSTRING
VAR_INPUT
	stKey: WSTRING;
END_VAR

IF stKey = "Company" THEN
	GetTextProperty := "Altus S.A.";
ELSIF stKey = "Project" THEN
	GetTextProperty := "NTP145_JIGA03_CPU_NX3030_0001";
ELSIF stKey = "Project Profile" THEN
	GetTextProperty := "Single";
ELSIF stKey = "Title" THEN
	GetTextProperty := "Super Teste NX3030";
ELSE
	GetTextProperty := "";
END_IF

END_FUNCTION

// Project Information/GetTextProperty2
// This function has been automatically generated from the project information.
{attribute 'signature_flag' := '1073741824'}
{attribute 'register_in_runtime'}
FUNCTION GetTextProperty2 : POINTER TO WSTRING
VAR_INPUT
	stKey: WSTRING;
END_VAR

IF stKey = "Company" THEN
	GetTextProperty2 := ADR("Altus S.A.");
ELSIF stKey = "Project" THEN
	GetTextProperty2 := ADR("NTP145_JIGA03_CPU_NX3030_0001");
ELSIF stKey = "Project Profile" THEN
	GetTextProperty2 := ADR("Single");
ELSIF stKey = "Title" THEN
	GetTextProperty2 := ADR("Super Teste NX3030");
ELSE
	GetTextProperty2 := ADR("");
END_IF

END_FUNCTION

// Project Information/GetNumberProperty
// This function has been automatically generated from the project information.
{attribute 'signature_flag' := '1073741824'}
{attribute 'register_in_runtime'}
FUNCTION GetNumberProperty : DINT
VAR_INPUT
	stKey: WSTRING;
END_VAR

GetNumberProperty := 0;

END_FUNCTION

// Project Information/GetBooleanProperty
// This function has been automatically generated from the project information.
{attribute 'signature_flag' := '1073741824'}
{attribute 'register_in_runtime'}
FUNCTION GetBooleanProperty : BOOL
VAR_INPUT
	stKey: WSTRING;
END_VAR

IF stKey = "Released" THEN
	GetBooleanProperty := FALSE;
ELSE
	GetBooleanProperty := FALSE;
END_IF

END_FUNCTION

// Project Information/GetVersionProperty
// This function has been automatically generated from the project information.
{attribute 'signature_flag' := '1073741824'}
{attribute 'register_in_runtime'}
FUNCTION GetVersionProperty : VERSION
VAR_INPUT
	stKey: WSTRING;
END_VAR

IF stKey = "Version" THEN
	GetVersionProperty.uiMajor := 3;
	GetVersionProperty.uiMinor := 61;
	GetVersionProperty.uiServicePack := 0;
	GetVersionProperty.uiPatch := 0;
ELSE
	GetVersionProperty.uiMajor := 0;
	GetVersionProperty.uiMinor := 0;
	GetVersionProperty.uiServicePack := 0;
	GetVersionProperty.uiPatch := 0;
END_IF

END_FUNCTION
